// TIA Portal project "Scambio_ferroviario2" (V15.1)

(* hardware
DEVICE "S7-1200 station_1"  S7-1200 Station
   slot 0: "Telaio di montaggio_0"  S7-1200 Rack  Rack  V1.0
   slot 1: "PLC_1"  CPU 1214C DC/DC/DC  6ES7 214-1AG40-0XB0  V4.2
*)

// ===== PLC "PLC_1"  CPU 1214C DC/DC/DC =====

VAR_GLOBAL   // PLC tag table "Tabella delle variabili standard"
   "P1" AT %I0.0 : Bool;
   "P2" AT %I0.1 : Bool;
   "SP1" AT %I0.2 : Bool;
   "SP2" AT %I0.3 : Bool;
   "SA1" AT %I0.4 : Bool;
   "SA2" AT %I0.5 : Bool;
   "A" AT %I0.6 : Bool;
   "B" AT %I0.7 : Bool;
   "C" AT %I1.0 : Bool;
   "D" AT %I1.1 : Bool;
   "S1" AT %Q0.0 : Bool;
   "D1" AT %Q0.1 : Bool;
   "S2" AT %Q0.2 : Bool;
   "D2" AT %Q0.3 : Bool;
   "SC1" AT %Q0.4 : Bool;
   "SC2" AT %Q0.5 : Bool;
   "semaforo" AT %M0.0 : Bool;
END_VAR

// folder: System blocks/Program resources

DATA_BLOCK "IEC_Timer_0_DB"   // DB1
{ S7_Optimized_Access := 'TRUE' }
AUTHOR : Simatic
FAMILY : IEC
NAME : IEC_TMR
VERSION : 1.0
// stored: InstanceOfName IEC_TIMER
"IEC_TIMER"
BEGIN
END_DATA_BLOCK

// folder: (top level)

FUNCTION_BLOCK "carrello"   // FB1, LAD
{ S7_Optimized_Access := 'TRUE' }
VERSION : 0.1
   VAR_INPUT
      FCP : Bool;
      FCA : Bool;
      partenza : Bool;
      fotocellulaArrivo : Bool;
      fotocellulaPartenza : Bool;
   END_VAR
   VAR_OUTPUT
      motore : Bool;
      SC1 : Bool;
      SC2 : Bool;
   END_VAR
   VAR RETAIN
      home : Bool := true;
      move1 : Bool;
      wait : Bool;
      move2 : Bool;
      move3 : Bool;
      attesaFine : Bool;
   END_VAR
   VAR CONSTANT
      tempo_attesa : Time := T#60s;
   END_VAR
BEGIN

REGION Network 1
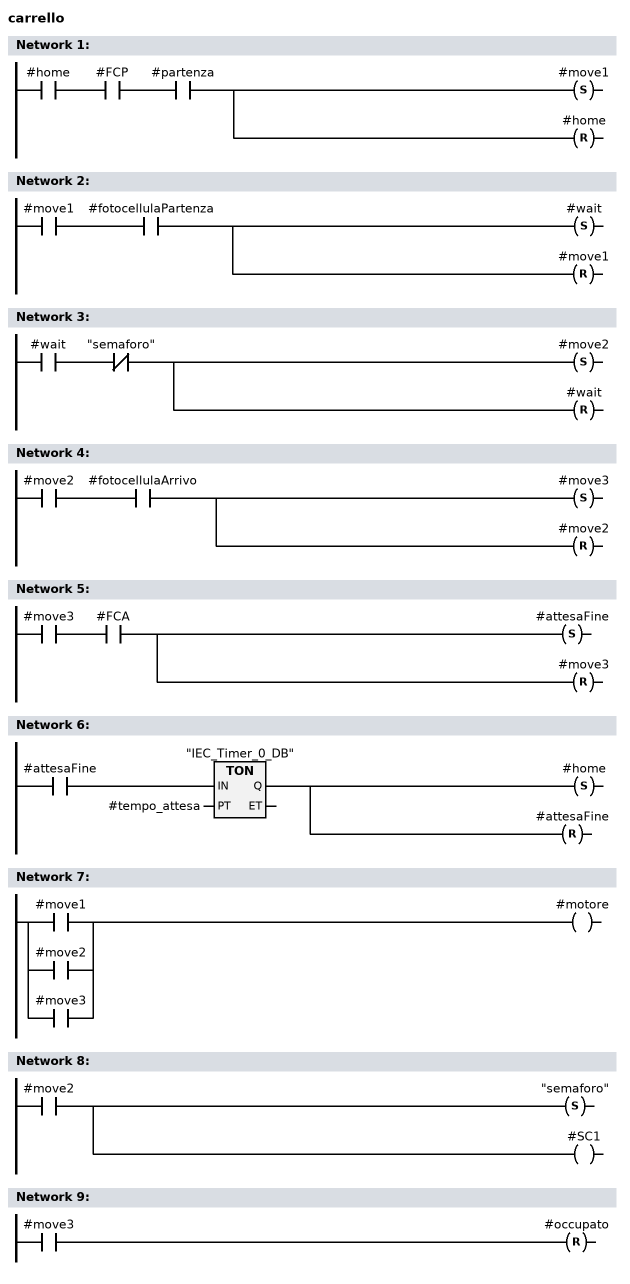
   RUNG wire#powerrail
      Contact( #home )
      Contact( #FCP )
      Contact( #partenza )
      wire#w1
      S_Coil( #move1 )
   END_RUNG
   RUNG wire#w1
      R_Coil( #home )
   END_RUNG
   // the same network as SCL:
   IF #home AND #FCP AND #partenza THEN
       #move1 := TRUE;
       #home := FALSE;
   END_IF;
END_REGION

REGION Network 2
   RUNG wire#powerrail
      Contact( #move1 )
      Contact( #fotocellulaPartenza )
      wire#w1
      S_Coil( #wait )
   END_RUNG
   RUNG wire#w1
      R_Coil( #move1 )
   END_RUNG
   // the same network as SCL:
   IF #move1 AND #fotocellulaPartenza THEN
       #wait := TRUE;
       #move1 := FALSE;
   END_IF;
END_REGION

REGION Network 3
   RUNG wire#powerrail
      Contact( #wait )
      I_Contact( "semaforo" )
      wire#w1
      S_Coil( #move2 )
   END_RUNG
   RUNG wire#w1
      R_Coil( #wait )
   END_RUNG
   // the same network as SCL:
   IF #wait AND NOT "semaforo" THEN
       #move2 := TRUE;
       #wait := FALSE;
   END_IF;
END_REGION

REGION Network 4
   RUNG wire#powerrail
      Contact( #move2 )
      Contact( #fotocellulaArrivo )
      wire#w1
      S_Coil( #move3 )
   END_RUNG
   RUNG wire#w1
      R_Coil( #move2 )
   END_RUNG
   // the same network as SCL:
   IF #move2 AND #fotocellulaArrivo THEN
       #move3 := TRUE;
       #move2 := FALSE;
   END_IF;
END_REGION

REGION Network 5
   RUNG wire#powerrail
      Contact( #move3 )
      Contact( #FCA )
      wire#w1
      S_Coil( #attesaFine )
   END_RUNG
   RUNG wire#w1
      R_Coil( #move3 )
   END_RUNG
   // the same network as SCL:
   IF #move3 AND #FCA THEN
       #attesaFine := TRUE;
       #move3 := FALSE;
   END_IF;
END_REGION

REGION Network 6
   "IEC_Timer_0_DB".TON(IN := #attesaFine, PT := #tempo_attesa);
   IF "IEC_Timer_0_DB".Q THEN
       #home := TRUE;
       #attesaFine := FALSE;
   END_IF;
END_REGION

REGION Network 7
   RUNG wire#powerrail
      Contact( #move1 )
      wire#w1
      Coil( #motore )
   END_RUNG
   RUNG wire#powerrail
      Contact( #move2 )
   END_RUNG wire#w1
   RUNG wire#powerrail
      Contact( #move3 )
   END_RUNG wire#w1
   // the same network as SCL:
   #motore := #move1 OR #move2 OR #move3;
END_REGION

REGION Network 8
   RUNG wire#powerrail
      Contact( #move2 )
      wire#w1
      S_Coil( "semaforo" )
   END_RUNG
   RUNG wire#w1
      Coil( #SC1 )
   END_RUNG
   // the same network as SCL:
   IF #move2 THEN "semaforo" := TRUE; END_IF;
   #SC1 := #move2;
END_REGION

REGION Network 9
   RUNG wire#powerrail
      Contact( #move3 )
      R_Coil( #occupato )
   END_RUNG
   // the same network as SCL:
   IF #move3 THEN #occupato := FALSE; END_IF;
END_REGION
END_FUNCTION_BLOCK

ORGANIZATION_BLOCK "Main"   // OB1, LAD, ProgramCycle
TITLE = "Main Program Sweep (Cycle)"
{ S7_Optimized_Access := 'TRUE' }
VERSION : 0.1
   VAR_INPUT
      Initial_Call : Bool;   // Initial call of this OB
      Remanence : Bool;   // =True, if remanent data are available
   END_VAR
BEGIN
END_ORGANIZATION_BLOCK